// TIA Portal V17 export
// export: Created 2025-01-08T13:55:34.3885705Z, ExportSetting WithDefaults, DisplayName Totally Integrated Automation Portal, DisplayVersion V17, DisplayName TIA Portal Openness, DisplayVersion V17, DisplayName TIA Portal Version Control Interface, DisplayVersion V17, DisplayName SINAMICS Startdrive Advanced, DisplayVersion V17 Update2, DisplayName SINAMICS Startdrive G130, G150, S120, S150, SINAMICS MV, S210, DisplayVersion V17 Update2, DisplayName SINAMICS Startdrive G110M, G120, G120C, G120D, G120P, G115D, DisplayVersion V17 Update2, DisplayName STEP 7 Professional, DisplayVersion V17, DisplayName STEP 7 Safety, DisplayVersion V17, DisplayName WinCC Advanced, DisplayVersion V17
DATA_BLOCK "FB - Speed_Changer_DB"   // DB4
VERSION : 0.1
// stored: AutoNumber true, DBAccessibleFromOPCUA true, DBAccessibleFromWebserver true, InstanceOfName FB - Speed_Changer, InstanceOfType FB
"FB - Speed_Changer"
   // VAR
   //    Speed_1_Pos : Bool;
   //    Speed_2_Pos : Bool;
   //    Speed_3_Pos : Bool;
   //    Speed_4_Pos : Bool;
   //    IEC_Timer_0_Instance { S7_SetPoint := 'True'} : TON_TIME;
   //    ResetSpeedEvents : Bool;
   //    Speed_5_Pos : Bool;
   // END_VAR
BEGIN
END_DATA_BLOCK
